FUNCTION HYST_1 (* Hystereses function *)
  (* Standard: 61499-1 *)
  (* Version 1.0, 2025-12-21, Franz Höpfinger *)
  PACKAGE OSCAT::Basic::POUs::Engineering::Control;
  IMPORT eclipse4diac::core::TypeHash;
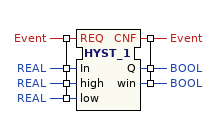
  EVENT_INPUT
    REQ WITH In, high, low;
  END_EVENT
  EVENT_OUTPUT
    CNF WITH Q, win;
  END_EVENT
  VAR_INPUT
    In : REAL;
    high : REAL;
    low : REAL;
  END_VAR
  VAR_OUTPUT
    Q : BOOL;
    win : BOOL;
  END_VAR
  BODY IN ST:
PACKAGE OSCAT::Basic::POUs::Engineering::Control;

(* Hystereses function *)
FUNCTION HYST_1
VAR_INPUT
	In : REAL;
	high : REAL;
	low : REAL;
END_VAR
VAR_OUTPUT
	Q : BOOL;
	win : BOOL;
END_VAR

(*
 * version 1.1	2. jun. 2008 programmer 	hugo tested BY	oscat
 * *
 * this hysteresis function switches the output high if the input signal reaches obove high and will
 * switch to low when the input falls back below low value.
 * a separate output mid is set if the input stays between low and high value.
 *)
IF In < low THEN
	Q := FALSE;
	win := FALSE;
ELSIF In > high THEN
	Q := TRUE;
	win := FALSE;
ELSE
	win := TRUE;
END_IF;

END_FUNCTION

(* revision history hm		4.  aug. 2006	rev 1.0 original version
 * *
 * hm		2. jun. 2008	rev 1.1 improved performance *)
  END_BODY
END_FUNCTION
